// TIA Portal project "Sistema_Irrigazione" (V15.1)

(* hardware
DEVICE "S7-1200 station_1"  S7-1200 Station
   slot 0: "Telaio di montaggio_0"  S7-1200 Rack  Rack  V1.0
   slot 1: "PLC_1"  CPU 1214C DC/DC/DC  6ES7 214-1AG40-0XB0  V4.2
*)

// ===== PLC "PLC_1"  CPU 1214C DC/DC/DC =====

VAR_GLOBAL   // PLC tag table "Tabella delle variabili standard"
   "SEC" AT %I0.0 : Bool;
   "apri_1" AT %Q0.0 : Bool;
   "apri_2" AT %Q0.1 : Bool;
   "chiudi_1" AT %Q0.2 : Bool;
   "chiudi_2" AT %Q0.3 : Bool;
END_VAR

VAR_GLOBAL CONSTANT   // PLC tag table "Tabella delle variabili standard"
   "apertura" : Time := T#40ms;
   "chiusura" : Time := T#20ms;
   "irrigazione" : Time := T#72h;
   "irrigazione_ramo" : Time := T#30s;
END_VAR

TYPE "VariabiliStato"
   STRUCT
      Home : Bool := true;
      Apri : Bool;
      Irriga : Bool;
      Chiudi : Bool;
   END_STRUCT;
END_TYPE

DATA_BLOCK "RamoIrrigazione1"   // DB1
{ S7_Optimized_Access := 'TRUE' }
VERSION : 0.1
// stored: InstanceOfName Funzione_irrigazione
"Funzione_irrigazione"
BEGIN
END_DATA_BLOCK

DATA_BLOCK "RamoIrrigazione2"   // DB2
{ S7_Optimized_Access := 'TRUE' }
VERSION : 0.1
// stored: InstanceOfName Funzione_irrigazione
"Funzione_irrigazione"
BEGIN
END_DATA_BLOCK

// folder: System blocks/Program resources

DATA_BLOCK "IntervalloIrrigazione"   // DB3
{ S7_Optimized_Access := 'TRUE' }
AUTHOR : Simatic
FAMILY : IEC
NAME : IEC_TMR
VERSION : 1.0
// stored: InstanceOfName IEC_TIMER
"IEC_TIMER"
BEGIN
END_DATA_BLOCK

// folder: (top level)

FUNCTION_BLOCK "Funzione_irrigazione"   // FB1, LAD
{ S7_Optimized_Access := 'TRUE' }
VERSION : 0.1
   VAR_INPUT
      abilita : Bool;
   END_VAR
   VAR_OUTPUT
      apri : Bool;
      chiudi : Bool := false;
   END_VAR
   VAR RETAIN
      Intervallo_apertura : TON_TIME;
      Intervallo_irrigazione : TON_TIME;
      Stato : "VariabiliStato";
      Intervallo_chiusura : TON_TIME;
   END_VAR
   VAR_TEMP   // added for the SCL form of the ladder/FBD networks
      _w1 : Bool;
   END_VAR
BEGIN

REGION Network 1
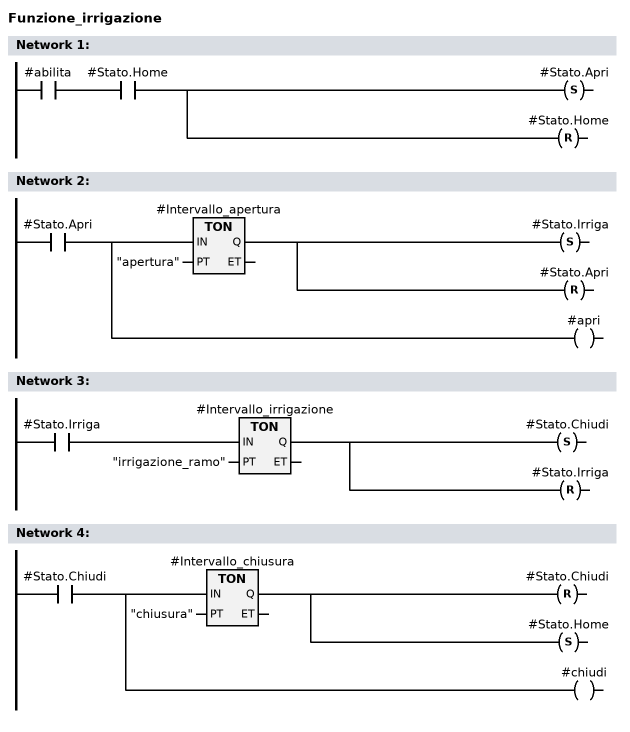
   RUNG wire#powerrail
      Contact( #abilita )
      Contact( #Stato.Home )
      wire#w1
      S_Coil( #Stato.Apri )
   END_RUNG
   RUNG wire#w1
      R_Coil( #Stato.Home )
   END_RUNG
   // the same network as SCL:
   IF #abilita AND #Stato.Home THEN
       #Stato.Apri := TRUE;
       #Stato.Home := FALSE;
   END_IF;
END_REGION

REGION Network 2
   #Intervallo_apertura(IN := #Stato.Apri, PT := "apertura");   // TON
   IF #Intervallo_apertura.Q THEN #Stato.Irriga := TRUE; END_IF;
   #_w1 := #Stato.Apri;
   IF #Intervallo_apertura.Q THEN #Stato.Apri := FALSE; END_IF;
   #apri := #_w1;
END_REGION

REGION Network 3
   #Intervallo_irrigazione(IN := #Stato.Irriga, PT := "irrigazione_ramo");   // TON
   IF #Intervallo_irrigazione.Q THEN
       #Stato.Chiudi := TRUE;
       #Stato.Irriga := FALSE;
   END_IF;
END_REGION

REGION Network 4
   #Intervallo_chiusura(IN := #Stato.Chiudi, PT := "chiusura");   // TON
   #_w1 := #Stato.Chiudi;
   IF #Intervallo_chiusura.Q THEN
       #Stato.Chiudi := FALSE;
       #Stato.Home := TRUE;
   END_IF;
   #chiudi := #_w1;
END_REGION
END_FUNCTION_BLOCK

ORGANIZATION_BLOCK "Main"   // OB1, LAD, ProgramCycle
TITLE = "Main Program Sweep (Cycle)"
{ S7_Optimized_Access := 'TRUE' }
VERSION : 0.1
   VAR_INPUT
      Initial_Call : Bool;   // Initial call of this OB
      Remanence : Bool;   // =True, if remanent data are available
   END_VAR
BEGIN

REGION Network 1
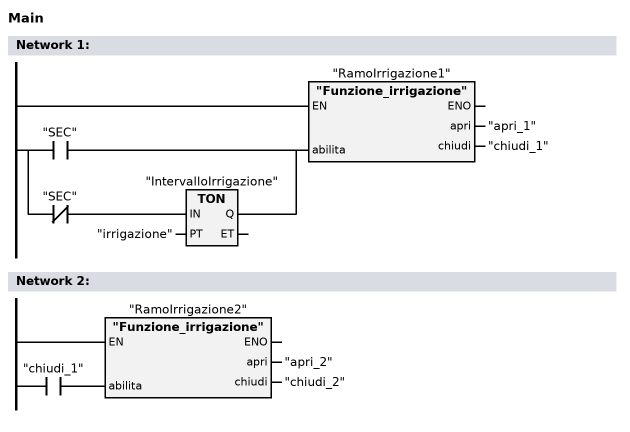
   "IntervalloIrrigazione".TON(IN := NOT "SEC", PT := "irrigazione");
   "RamoIrrigazione1"(abilita := "SEC" OR "IntervalloIrrigazione".Q, apri => "apri_1", chiudi => "chiudi_1");   // "Funzione_irrigazione"
END_REGION

REGION Network 2
   RUNG wire#powerrail
      "RamoIrrigazione2"(abilita := wire#w1, apri => "apri_2", chiudi => "chiudi_2")
   END_RUNG
   RUNG wire#powerrail
      Contact( "chiudi_1" )
   END_RUNG wire#w1
   // the same network as SCL:
   "RamoIrrigazione2"(abilita := "chiudi_1", apri => "apri_2", chiudi => "chiudi_2");   // "Funzione_irrigazione"
END_REGION
END_ORGANIZATION_BLOCK